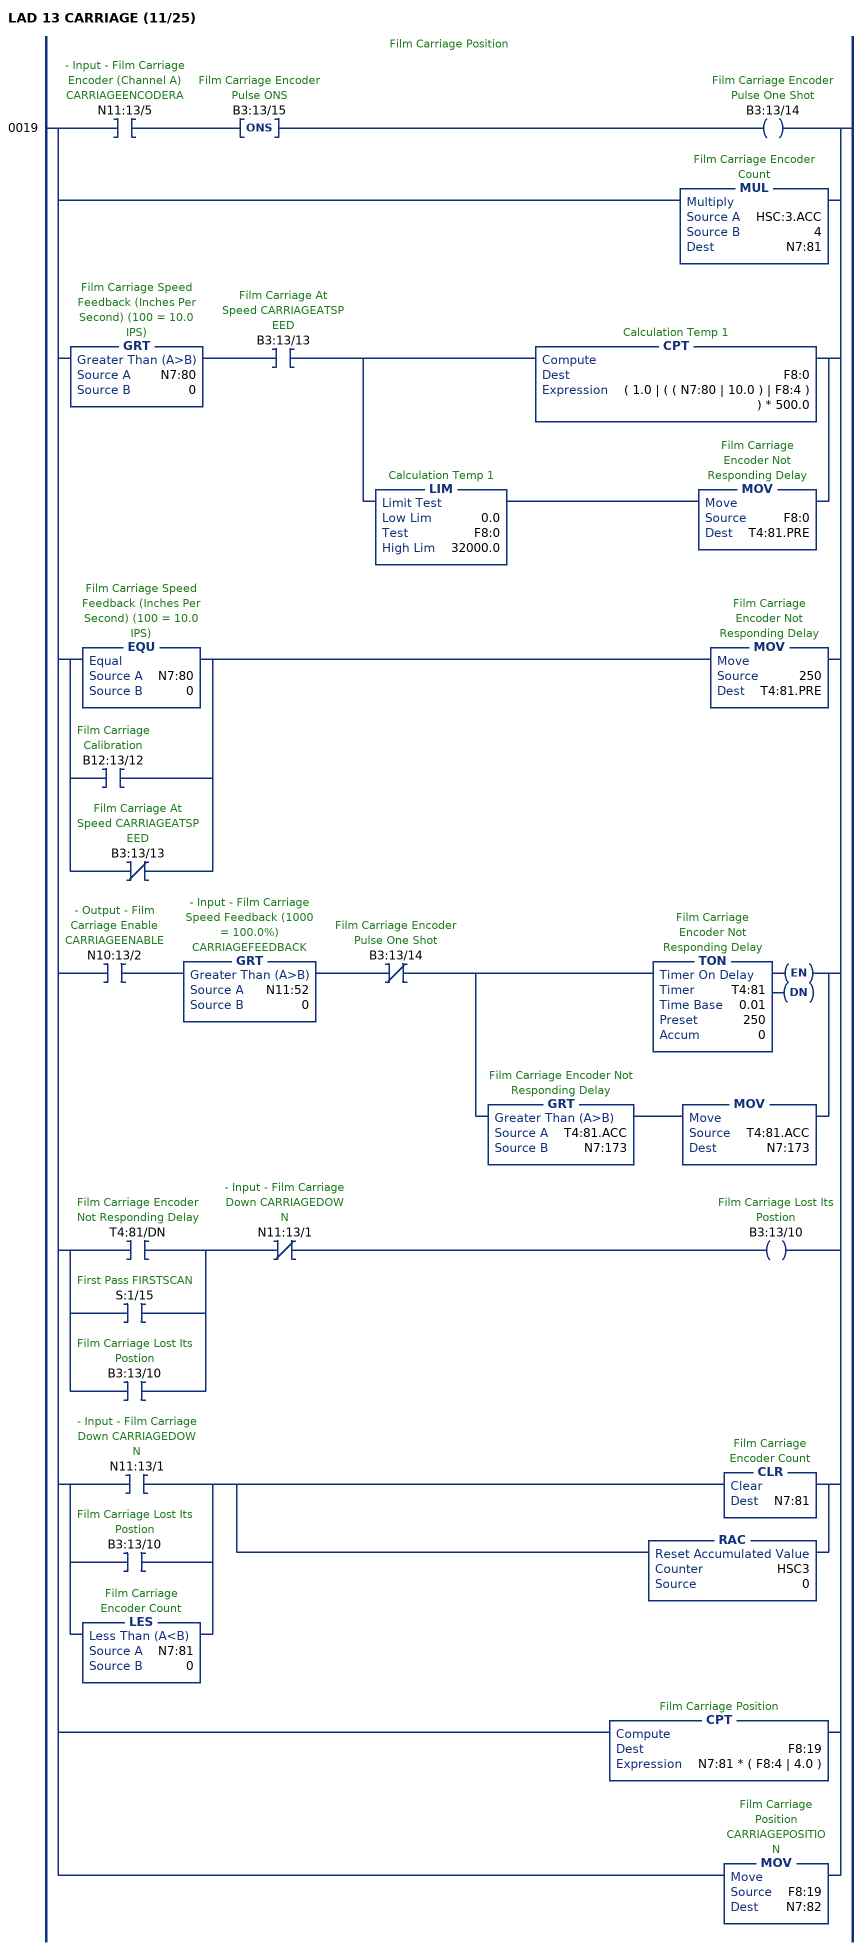
% Rung: 19 %
% Film Carriage Position %
SOR BST XIC N11:13/5 ONS B3:13/15 OTE B3:13/14 NXB MUL HSC:3.ACC 4 N7:81 NXB BST GRT N7:80 0 XIC B3:13/13 BST CPT F8:0 " ( 1.0 | ( ( N7:80 | 10.0 ) | F8:4 ) ) * 500.0 " NXB LIM 0.0 F8:0 32000.0 MOV F8:0 T4:81.PRE BND NXB BST EQU N7:80 0 NXB XIC B12:13/12 NXB XIO B3:13/13 BND MOV 250 T4:81.PRE BND NXB XIC N10:13/2 GRT N11:52 0 XIO B3:13/14 BST TON T4:81 0.01 250 0 NXB GRT T4:81.ACC N7:173 MOV T4:81.ACC N7:173 BND NXB BST XIC T4:81/DN NXB XIC S:1/15 NXB XIC B3:13/10 BND XIO N11:13/1 OTE B3:13/10 NXB BST XIC N11:13/1 NXB XIC B3:13/10 NXB LES N7:81 0 BND BST CLR N7:81 NXB RAC HSC3 0 BND NXB CPT F8:19 " N7:81 * ( F8:4 | 4.0 ) " NXB MOV F8:19 N7:82 BND EOR
%   N11:13/5  CARRIAGEENCODERA  "- Input - Film Carriage Encoder (Channel A)" %
%   B3:13/15  "Film Carriage Encoder Pulse ONS" %
%   B3:13/14  "Film Carriage Encoder Pulse One Shot" %
%   N7:81  "Film Carriage Encoder Count" %
%   N7:80  "Film Carriage Speed Feedback (Inches Per Second) (100 = 10.0 IPS)" %
%   B3:13/13  CARRIAGEATSPEED  "Film Carriage At Speed" %
%   F8:0  "Calculation Temp 1" %
%   F8:4  CARRIAGEENCODERRES  "Film Carriage Encoder Resolution (Inches Per Pulse)" %
%   T4:81  "Film Carriage Encoder Not Responding Delay" %
%   B12:13/12  "Film Carriage Calibration" %
%   N10:13/2  CARRIAGEENABLE  "- Output - Film Carriage Enable" %
%   N11:52  CARRIAGEFEEDBACK  "- Input - Film Carriage Speed Feedback (1000 = 100.0%)" %
%   S:1/15  FIRSTSCAN  "First Pass" %
%   B3:13/10  "Film Carriage Lost Its Postion" %
%   N11:13/1  CARRIAGEDOWN  "- Input - Film Carriage Down" %
%   F8:19  "Film Carriage Position" %
%   N7:82  CARRIAGEPOSITION  "Film Carriage Position" %

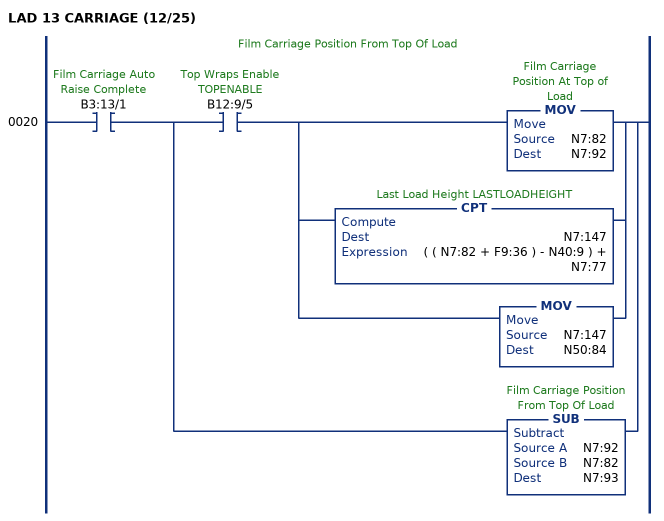
% Rung: 20 %
% Film Carriage Position From Top Of Load %
SOR XIC B3:13/1 BST XIC B12:9/5 BST MOV N7:82 N7:92 NXB CPT N7:147 " ( ( N7:82 + F9:36 ) - N40:9 ) + N7:77 " NXB MOV N7:147 N50:84 BND NXB SUB N7:92 N7:82 N7:93 BND EOR
%   B3:13/1  "Film Carriage Auto Raise Complete" %
%   B12:9/5  TOPENABLE  "Top Wraps Enable" %
%   N7:82  CARRIAGEPOSITION  "Film Carriage Position" %
%   N7:92  "Film Carriage Position At Top of Load" %
%   N7:147  LASTLOADHEIGHT  "Last Load Height" %
%   F9:36  FILMWIDTHATLOAD  "Film Width At Load" %
%   N40:9  "Current Profile Top Overwrap (Inches)" %
%   N7:77  "Carriage Pallet Grip Drive Down" %
%   N7:93  "Film Carriage Position From Top Of Load" %

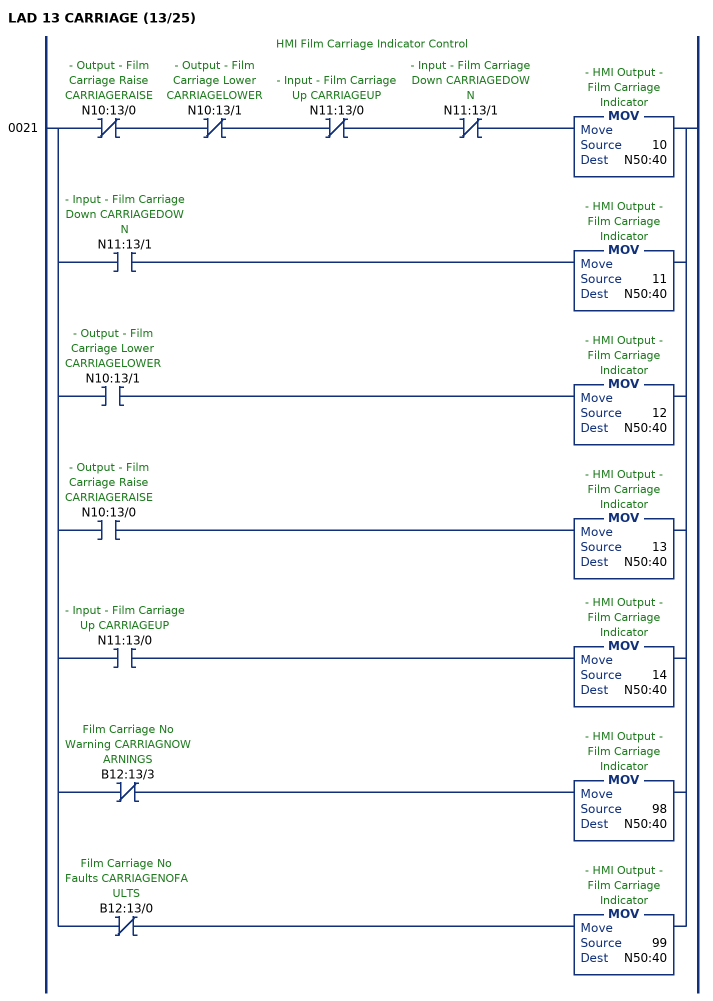
% Rung: 21 %
% HMI Film Carriage Indicator Control %
SOR BST XIO N10:13/0 XIO N10:13/1 XIO N11:13/0 XIO N11:13/1 MOV 10 N50:40 NXB XIC N11:13/1 MOV 11 N50:40 NXB XIC N10:13/1 MOV 12 N50:40 NXB XIC N10:13/0 MOV 13 N50:40 NXB XIC N11:13/0 MOV 14 N50:40 NXB XIO B12:13/3 MOV 98 N50:40 NXB XIO B12:13/0 MOV 99 N50:40 BND EOR
%   N10:13/0  CARRIAGERAISE  "- Output - Film Carriage Raise" %
%   N10:13/1  CARRIAGELOWER  "- Output - Film Carriage Lower" %
%   N11:13/0  CARRIAGEUP  "- Input - Film Carriage Up" %
%   N11:13/1  CARRIAGEDOWN  "- Input - Film Carriage Down" %
%   N50:40  "- HMI Output - Film Carriage Indicator" %
%   B12:13/3  CARRIAGNOWARNINGS  "Film Carriage No Warning" %
%   B12:13/0  CARRIAGENOFAULTS  "Film Carriage No Faults" %

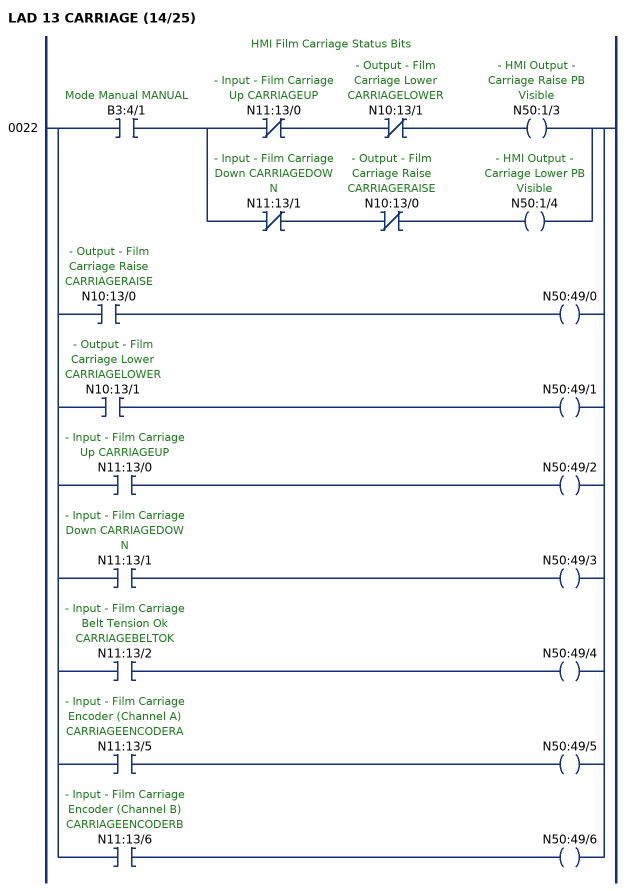
% Rung: 22 %
% HMI Film Carriage Status Bits %
SOR BST XIC B3:4/1 BST XIO N11:13/0 XIO N10:13/1 OTE N50:1/3 NXB XIO N11:13/1 XIO N10:13/0 OTE N50:1/4 BND NXB XIC N10:13/0 OTE N50:49/0 NXB XIC N10:13/1 OTE N50:49/1 NXB XIC N11:13/0 OTE N50:49/2 NXB XIC N11:13/1 OTE N50:49/3 NXB XIC N11:13/2 OTE N50:49/4 NXB XIC N11:13/5 OTE N50:49/5 NXB XIC N11:13/6 OTE N50:49/6 BND EOR
%   B3:4/1  MANUAL  "Mode Manual" %
%   N11:13/0  CARRIAGEUP  "- Input - Film Carriage Up" %
%   N10:13/1  CARRIAGELOWER  "- Output - Film Carriage Lower" %
%   N50:1/3  "- HMI Output - Carriage Raise PB Visible" %
%   N11:13/1  CARRIAGEDOWN  "- Input - Film Carriage Down" %
%   N10:13/0  CARRIAGERAISE  "- Output - Film Carriage Raise" %
%   N50:1/4  "- HMI Output - Carriage Lower PB Visible" %
%   N11:13/2  CARRIAGEBELTOK  "- Input - Film Carriage Belt Tension Ok" %
%   N11:13/5  CARRIAGEENCODERA  "- Input - Film Carriage Encoder (Channel A)" %
%   N11:13/6  CARRIAGEENCODERB  "- Input - Film Carriage Encoder (Channel B)" %

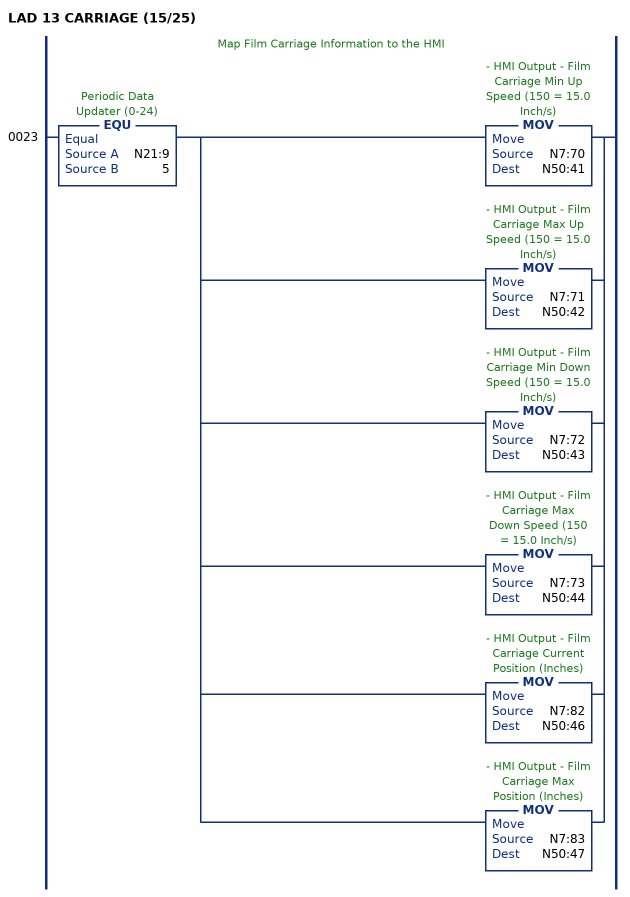
% Rung: 23 %
% Map Film Carriage Information to the HMI %
SOR EQU N21:9 5 BST MOV N7:70 N50:41 NXB MOV N7:71 N50:42 NXB MOV N7:72 N50:43 NXB MOV N7:73 N50:44 NXB MOV N7:82 N50:46 NXB MOV N7:83 N50:47 BND EOR
%   N21:9  "Periodic Data Updater (0-24)" %
%   N7:70  "Film Carriage Up Min Speed (Inches Per Second) (100 = 10.0 IPS)" %
%   N50:41  "- HMI Output - Film Carriage Min Up Speed (150 = 15.0 Inch/s)" %
%   N7:71  "Film Carriage Up Max Speed (Inches Per Second) (100 = 10.0 IPS)" %
%   N50:42  "- HMI Output - Film Carriage Max Up Speed (150 = 15.0 Inch/s)" %
%   N7:72  "Film Carriage Down Min Speed (Inches Per Second) (100 = 10.0 IPS)" %
%   N50:43  "- HMI Output - Film Carriage Min Down Speed (150 = 15.0 Inch/s)" %
%   N7:73  "Film Carriage Down Max Speed (Inches Per Second) (100 = 10.0 IPS)" %
%   N50:44  "- HMI Output - Film Carriage Max Down Speed (150 = 15.0 Inch/s)" %
%   N7:82  CARRIAGEPOSITION  "Film Carriage Position" %
%   N50:46  "- HMI Output - Film Carriage Current Position (Inches)" %
%   N7:83  CARRIAGEMAXPOSITION  "Film Carriage Max Position" %
%   N50:47  "- HMI Output - Film Carriage Max Position (Inches)" %

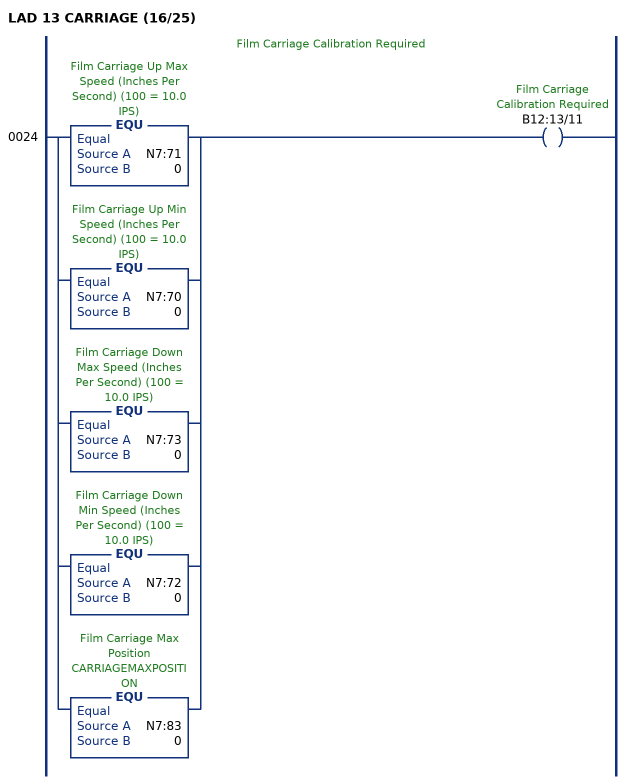
% Rung: 24 %
% Film Carriage Calibration Required %
SOR BST EQU N7:71 0 NXB EQU N7:70 0 NXB EQU N7:73 0 NXB EQU N7:72 0 NXB EQU N7:83 0 BND OTE B12:13/11 EOR
%   N7:71  "Film Carriage Up Max Speed (Inches Per Second) (100 = 10.0 IPS)" %
%   N7:70  "Film Carriage Up Min Speed (Inches Per Second) (100 = 10.0 IPS)" %
%   N7:73  "Film Carriage Down Max Speed (Inches Per Second) (100 = 10.0 IPS)" %
%   N7:72  "Film Carriage Down Min Speed (Inches Per Second) (100 = 10.0 IPS)" %
%   N7:83  CARRIAGEMAXPOSITION  "Film Carriage Max Position" %
%   B12:13/11  "Film Carriage Calibration Required" %

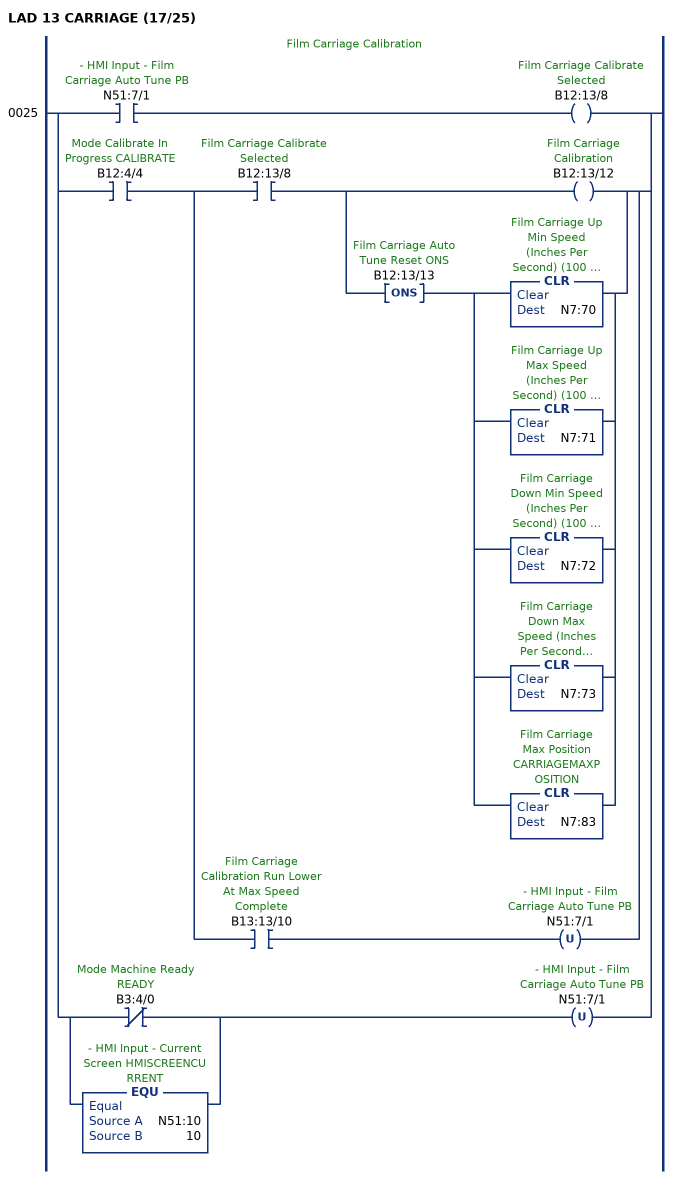
% Rung: 25 %
% Film Carriage Calibration %
SOR BST XIC N51:7/1 OTE B12:13/8 NXB XIC B12:4/4 BST XIC B12:13/8 BST OTE B12:13/12 NXB ONS B12:13/13 BST CLR N7:70 NXB CLR N7:71 NXB CLR N7:72 NXB CLR N7:73 NXB CLR N7:83 BND BND NXB XIC B13:13/10 OTU N51:7/1 BND NXB BST XIO B3:4/0 NXB EQU N51:10 10 BND OTU N51:7/1 BND EOR
%   N51:7/1  "- HMI Input - Film Carriage Auto Tune PB" %
%   B12:13/8  "Film Carriage Calibrate Selected" %
%   B12:4/4  CALIBRATE  "Mode Calibrate In Progress" %
%   B12:13/12  "Film Carriage Calibration" %
%   B12:13/13  "Film Carriage Auto Tune Reset ONS" %
%   N7:70  "Film Carriage Up Min Speed (Inches Per Second) (100 = 10.0 IPS)" %
%   N7:71  "Film Carriage Up Max Speed (Inches Per Second) (100 = 10.0 IPS)" %
%   N7:72  "Film Carriage Down Min Speed (Inches Per Second) (100 = 10.0 IPS)" %
%   N7:73  "Film Carriage Down Max Speed (Inches Per Second) (100 = 10.0 IPS)" %
%   N7:83  CARRIAGEMAXPOSITION  "Film Carriage Max Position" %
%   B13:13/10  "Film Carriage Calibration Run Lower At Max Speed Complete" %
%   B3:4/0  READY  "Mode Machine Ready" %
%   N51:10  HMISCREENCURRENT  "- HMI Input - Current Screen" %

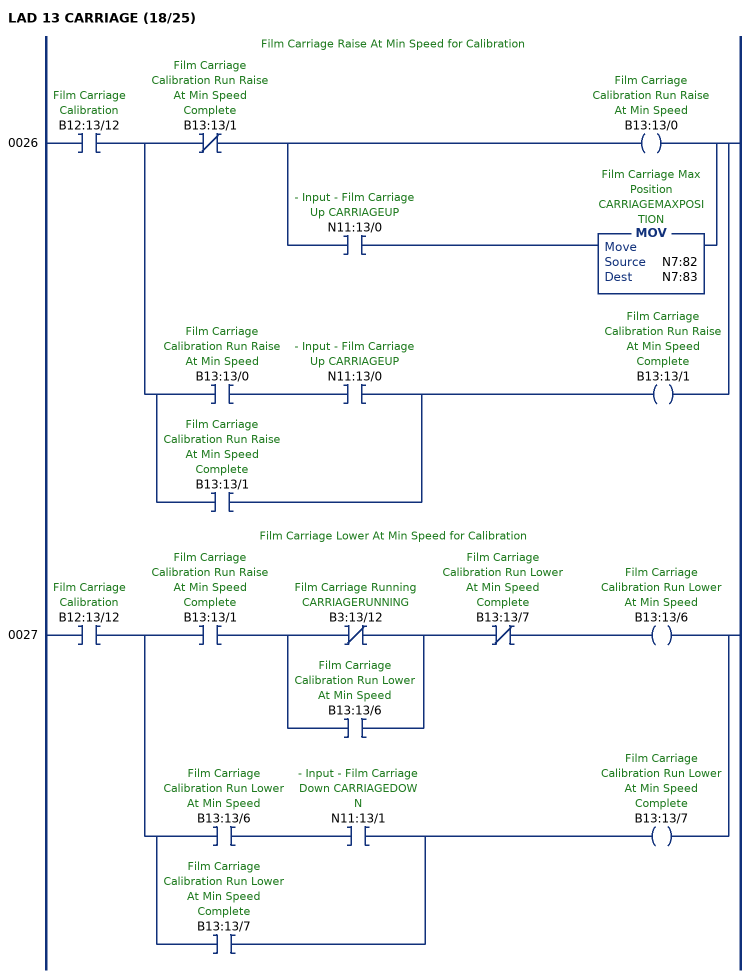
% Rung: 26 %
% Film Carriage Raise At Min Speed for Calibration %
SOR XIC B12:13/12 BST XIO B13:13/1 BST OTE B13:13/0 NXB XIC N11:13/0 MOV N7:82 N7:83 BND NXB BST XIC B13:13/0 XIC N11:13/0 NXB XIC B13:13/1 BND OTE B13:13/1 BND EOR
%   B12:13/12  "Film Carriage Calibration" %
%   B13:13/1  "Film Carriage Calibration Run Raise At Min Speed Complete" %
%   B13:13/0  "Film Carriage Calibration Run Raise At Min Speed" %
%   N11:13/0  CARRIAGEUP  "- Input - Film Carriage Up" %
%   N7:82  CARRIAGEPOSITION  "Film Carriage Position" %
%   N7:83  CARRIAGEMAXPOSITION  "Film Carriage Max Position" %
% Rung: 27 %
% Film Carriage Lower At Min Speed for Calibration %
SOR XIC B12:13/12 BST XIC B13:13/1 BST XIO B3:13/12 NXB XIC B13:13/6 BND XIO B13:13/7 OTE B13:13/6 NXB BST XIC B13:13/6 XIC N11:13/1 NXB XIC B13:13/7 BND OTE B13:13/7 BND EOR
%   B12:13/12  "Film Carriage Calibration" %
%   B13:13/1  "Film Carriage Calibration Run Raise At Min Speed Complete" %
%   B3:13/12  CARRIAGERUNNING  "Film Carriage Running" %
%   B13:13/6  "Film Carriage Calibration Run Lower At Min Speed" %
%   B13:13/7  "Film Carriage Calibration Run Lower At Min Speed Complete" %
%   N11:13/1  CARRIAGEDOWN  "- Input - Film Carriage Down" %

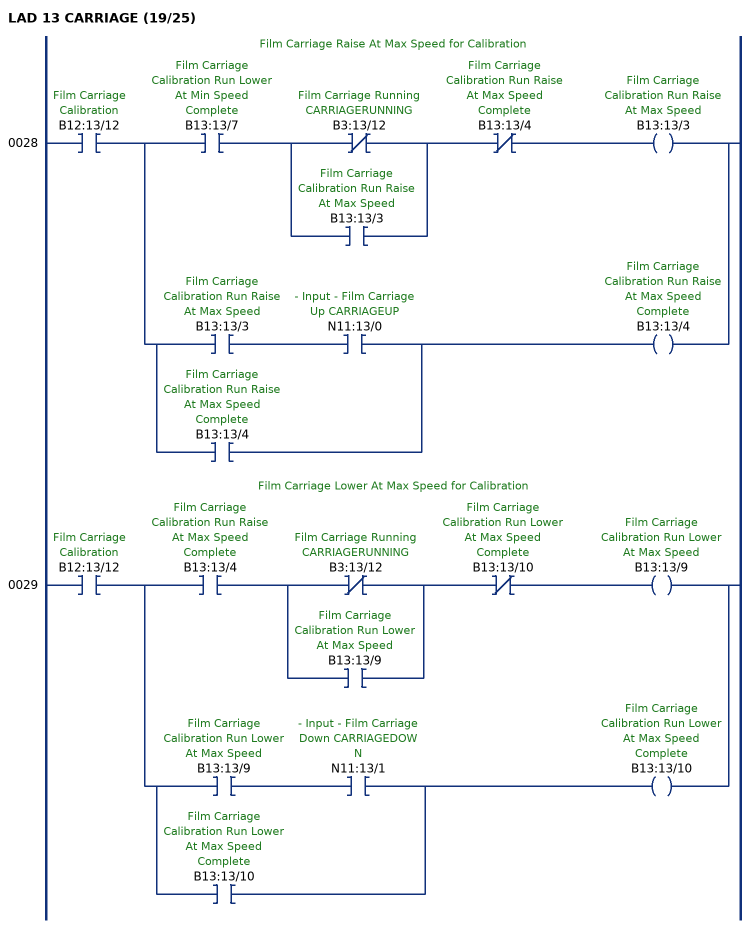
% Rung: 28 %
% Film Carriage Raise At Max Speed for Calibration %
SOR XIC B12:13/12 BST XIC B13:13/7 BST XIO B3:13/12 NXB XIC B13:13/3 BND XIO B13:13/4 OTE B13:13/3 NXB BST XIC B13:13/3 XIC N11:13/0 NXB XIC B13:13/4 BND OTE B13:13/4 BND EOR
%   B12:13/12  "Film Carriage Calibration" %
%   B13:13/7  "Film Carriage Calibration Run Lower At Min Speed Complete" %
%   B3:13/12  CARRIAGERUNNING  "Film Carriage Running" %
%   B13:13/3  "Film Carriage Calibration Run Raise At Max Speed" %
%   B13:13/4  "Film Carriage Calibration Run Raise At Max Speed Complete" %
%   N11:13/0  CARRIAGEUP  "- Input - Film Carriage Up" %
% Rung: 29 %
% Film Carriage Lower At Max Speed for Calibration %
SOR XIC B12:13/12 BST XIC B13:13/4 BST XIO B3:13/12 NXB XIC B13:13/9 BND XIO B13:13/10 OTE B13:13/9 NXB BST XIC B13:13/9 XIC N11:13/1 NXB XIC B13:13/10 BND OTE B13:13/10 BND EOR
%   B12:13/12  "Film Carriage Calibration" %
%   B13:13/4  "Film Carriage Calibration Run Raise At Max Speed Complete" %
%   B3:13/12  CARRIAGERUNNING  "Film Carriage Running" %
%   B13:13/9  "Film Carriage Calibration Run Lower At Max Speed" %
%   B13:13/10  "Film Carriage Calibration Run Lower At Max Speed Complete" %
%   N11:13/1  CARRIAGEDOWN  "- Input - Film Carriage Down" %

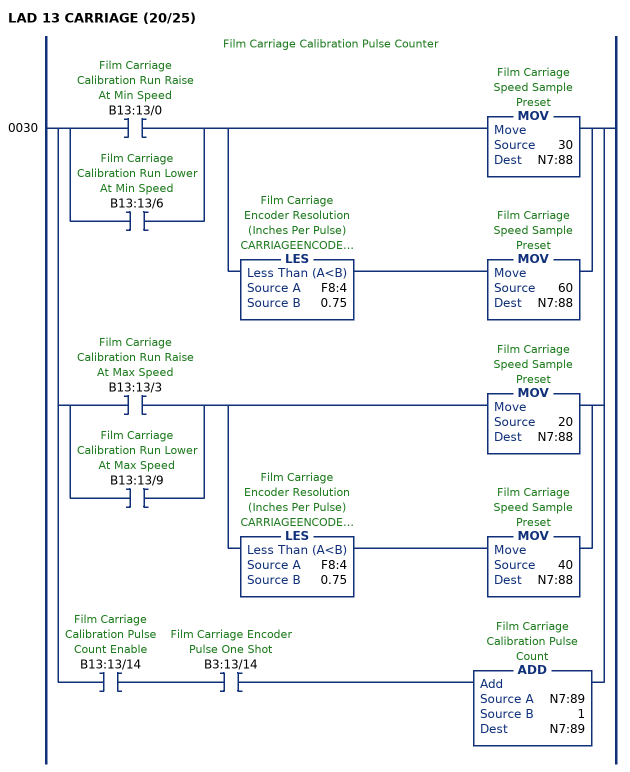
% Rung: 30 %
% Film Carriage Calibration Pulse Counter %
SOR BST BST XIC B13:13/0 NXB XIC B13:13/6 BND BST MOV 30 N7:88 NXB LES F8:4 0.75 MOV 60 N7:88 BND NXB BST XIC B13:13/3 NXB XIC B13:13/9 BND BST MOV 20 N7:88 NXB LES F8:4 0.75 MOV 40 N7:88 BND NXB XIC B13:13/14 XIC B3:13/14 ADD N7:89 1 N7:89 BND EOR
%   B13:13/0  "Film Carriage Calibration Run Raise At Min Speed" %
%   B13:13/6  "Film Carriage Calibration Run Lower At Min Speed" %
%   N7:88  "Film Carriage Speed Sample Preset" %
%   F8:4  CARRIAGEENCODERRES  "Film Carriage Encoder Resolution (Inches Per Pulse)" %
%   B13:13/3  "Film Carriage Calibration Run Raise At Max Speed" %
%   B13:13/9  "Film Carriage Calibration Run Lower At Max Speed" %
%   B13:13/14  "Film Carriage Calibration Pulse Count Enable" %
%   B3:13/14  "Film Carriage Encoder Pulse One Shot" %
%   N7:89  "Film Carriage Calibration Pulse Count" %

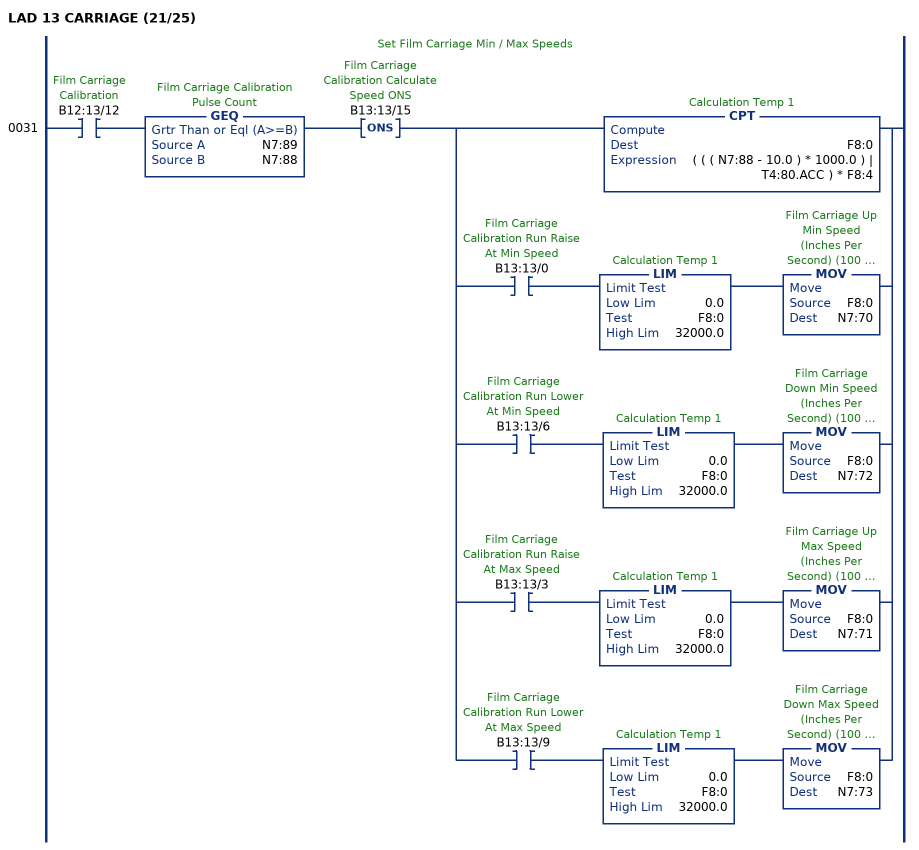
% Rung: 31 %
% Set Film Carriage Min / Max Speeds %
SOR XIC B12:13/12 GEQ N7:89 N7:88 ONS B13:13/15 BST CPT F8:0 " ( ( ( N7:88 - 10.0 ) * 1000.0 ) | T4:80.ACC ) * F8:4 " NXB XIC B13:13/0 LIM 0.0 F8:0 32000.0 MOV F8:0 N7:70 NXB XIC B13:13/6 LIM 0.0 F8:0 32000.0 MOV F8:0 N7:72 NXB XIC B13:13/3 LIM 0.0 F8:0 32000.0 MOV F8:0 N7:71 NXB XIC B13:13/9 LIM 0.0 F8:0 32000.0 MOV F8:0 N7:73 BND EOR
%   B12:13/12  "Film Carriage Calibration" %
%   N7:89  "Film Carriage Calibration Pulse Count" %
%   N7:88  "Film Carriage Speed Sample Preset" %
%   B13:13/15  "Film Carriage Calibration Calculate Speed ONS" %
%   F8:0  "Calculation Temp 1" %
%   T4:80  "Film Carriage Calibration Time" %
%   F8:4  CARRIAGEENCODERRES  "Film Carriage Encoder Resolution (Inches Per Pulse)" %
%   B13:13/0  "Film Carriage Calibration Run Raise At Min Speed" %
%   N7:70  "Film Carriage Up Min Speed (Inches Per Second) (100 = 10.0 IPS)" %
%   B13:13/6  "Film Carriage Calibration Run Lower At Min Speed" %
%   N7:72  "Film Carriage Down Min Speed (Inches Per Second) (100 = 10.0 IPS)" %
%   B13:13/3  "Film Carriage Calibration Run Raise At Max Speed" %
%   N7:71  "Film Carriage Up Max Speed (Inches Per Second) (100 = 10.0 IPS)" %
%   B13:13/9  "Film Carriage Calibration Run Lower At Max Speed" %
%   N7:73  "Film Carriage Down Max Speed (Inches Per Second) (100 = 10.0 IPS)" %

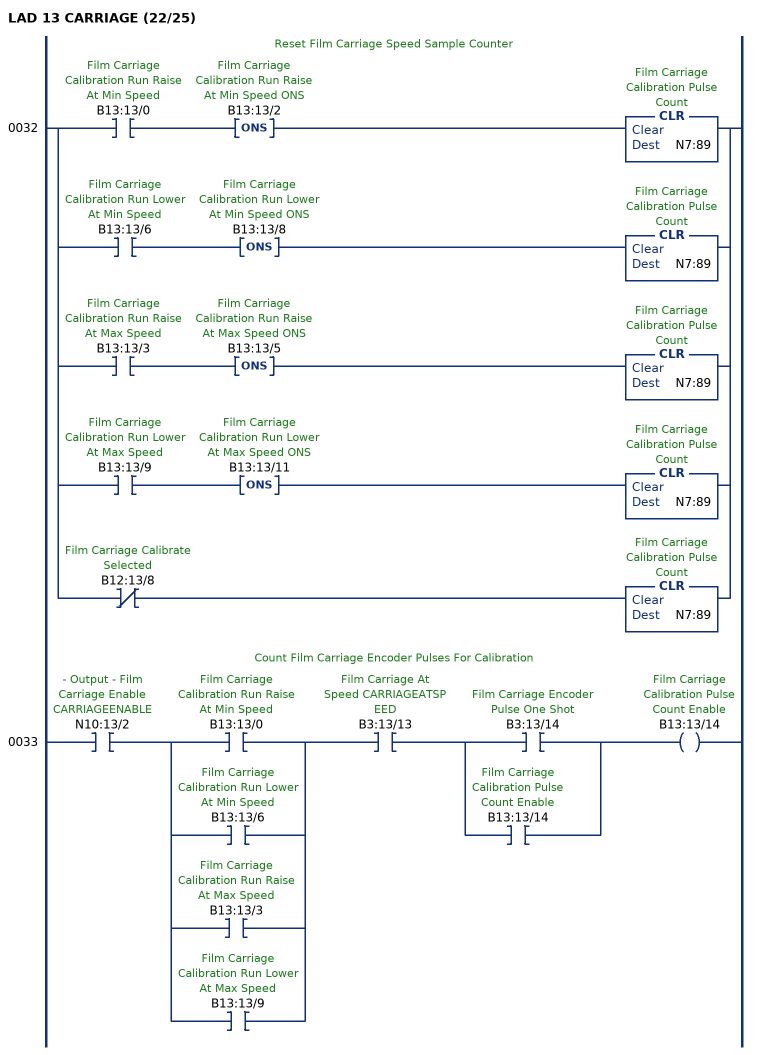
% Rung: 32 %
% Reset Film Carriage Speed Sample Counter %
SOR BST XIC B13:13/0 ONS B13:13/2 CLR N7:89 NXB XIC B13:13/6 ONS B13:13/8 CLR N7:89 NXB XIC B13:13/3 ONS B13:13/5 CLR N7:89 NXB XIC B13:13/9 ONS B13:13/11 CLR N7:89 NXB XIO B12:13/8 CLR N7:89 BND EOR
%   B13:13/0  "Film Carriage Calibration Run Raise At Min Speed" %
%   B13:13/2  "Film Carriage Calibration Run Raise At Min Speed ONS" %
%   N7:89  "Film Carriage Calibration Pulse Count" %
%   B13:13/6  "Film Carriage Calibration Run Lower At Min Speed" %
%   B13:13/8  "Film Carriage Calibration Run Lower At Min Speed ONS" %
%   B13:13/3  "Film Carriage Calibration Run Raise At Max Speed" %
%   B13:13/5  "Film Carriage Calibration Run Raise At Max Speed ONS" %
%   B13:13/9  "Film Carriage Calibration Run Lower At Max Speed" %
%   B13:13/11  "Film Carriage Calibration Run Lower At Max Speed ONS" %
%   B12:13/8  "Film Carriage Calibrate Selected" %
% Rung: 33 %
% Count Film Carriage Encoder Pulses For Calibration %
SOR XIC N10:13/2 BST XIC B13:13/0 NXB XIC B13:13/6 NXB XIC B13:13/3 NXB XIC B13:13/9 BND XIC B3:13/13 BST XIC B3:13/14 NXB XIC B13:13/14 BND OTE B13:13/14 EOR
%   N10:13/2  CARRIAGEENABLE  "- Output - Film Carriage Enable" %
%   B13:13/0  "Film Carriage Calibration Run Raise At Min Speed" %
%   B13:13/6  "Film Carriage Calibration Run Lower At Min Speed" %
%   B13:13/3  "Film Carriage Calibration Run Raise At Max Speed" %
%   B13:13/9  "Film Carriage Calibration Run Lower At Max Speed" %
%   B3:13/13  CARRIAGEATSPEED  "Film Carriage At Speed" %
%   B3:13/14  "Film Carriage Encoder Pulse One Shot" %
%   B13:13/14  "Film Carriage Calibration Pulse Count Enable" %

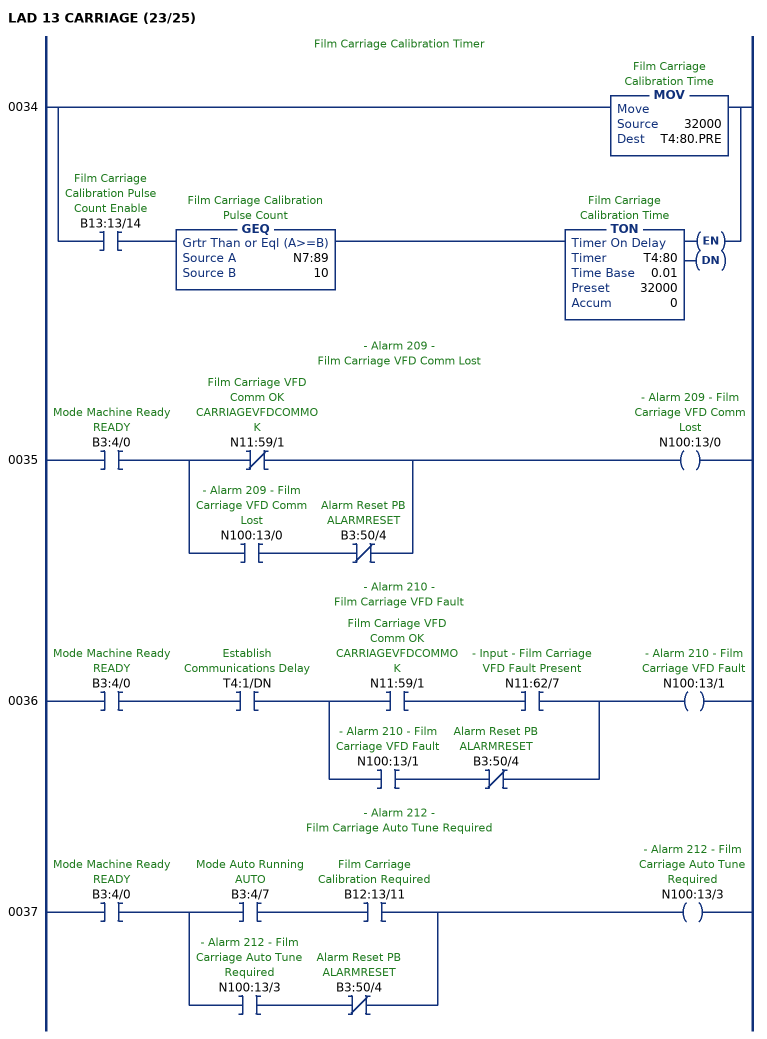
% Rung: 34 %
% Film Carriage Calibration Timer %
SOR BST MOV 32000 T4:80.PRE NXB XIC B13:13/14 GEQ N7:89 10 TON T4:80 0.01 32000 0 BND EOR
%   T4:80  "Film Carriage Calibration Time" %
%   B13:13/14  "Film Carriage Calibration Pulse Count Enable" %
%   N7:89  "Film Carriage Calibration Pulse Count" %
% Rung: 35 %
% - Alarm 209 -
% 
% Film Carriage VFD Comm Lost %
SOR XIC B3:4/0 BST XIO N11:59/1 NXB XIC N100:13/0 XIO B3:50/4 BND OTE N100:13/0 EOR
%   B3:4/0  READY  "Mode Machine Ready" %
%   N11:59/1  CARRIAGEVFDCOMMOK  "Film Carriage VFD Comm OK" %
%   N100:13/0  "- Alarm 209 - Film Carriage VFD Comm Lost" %
%   B3:50/4  ALARMRESET  "Alarm Reset PB" %
% Rung: 36 %
% - Alarm 210 -
% 
% Film Carriage VFD Fault %
SOR XIC B3:4/0 XIC T4:1/DN BST XIC N11:59/1 XIC N11:62/7 NXB XIC N100:13/1 XIO B3:50/4 BND OTE N100:13/1 EOR
%   B3:4/0  READY  "Mode Machine Ready" %
%   T4:1  "Establish Communications Delay" %
%   N11:59/1  CARRIAGEVFDCOMMOK  "Film Carriage VFD Comm OK" %
%   N11:62/7  "- Input - Film Carriage VFD Fault Present" %
%   N100:13/1  "- Alarm 210 - Film Carriage VFD Fault" %
%   B3:50/4  ALARMRESET  "Alarm Reset PB" %
% Rung: 37 %
% - Alarm 212 -
% 
% Film Carriage Auto Tune Required %
SOR XIC B3:4/0 BST XIC B3:4/7 XIC B12:13/11 NXB XIC N100:13/3 XIO B3:50/4 BND OTE N100:13/3 EOR
%   B3:4/0  READY  "Mode Machine Ready" %
%   B3:4/7  AUTO  "Mode Auto Running" %
%   B12:13/11  "Film Carriage Calibration Required" %
%   N100:13/3  "- Alarm 212 - Film Carriage Auto Tune Required" %
%   B3:50/4  ALARMRESET  "Alarm Reset PB" %

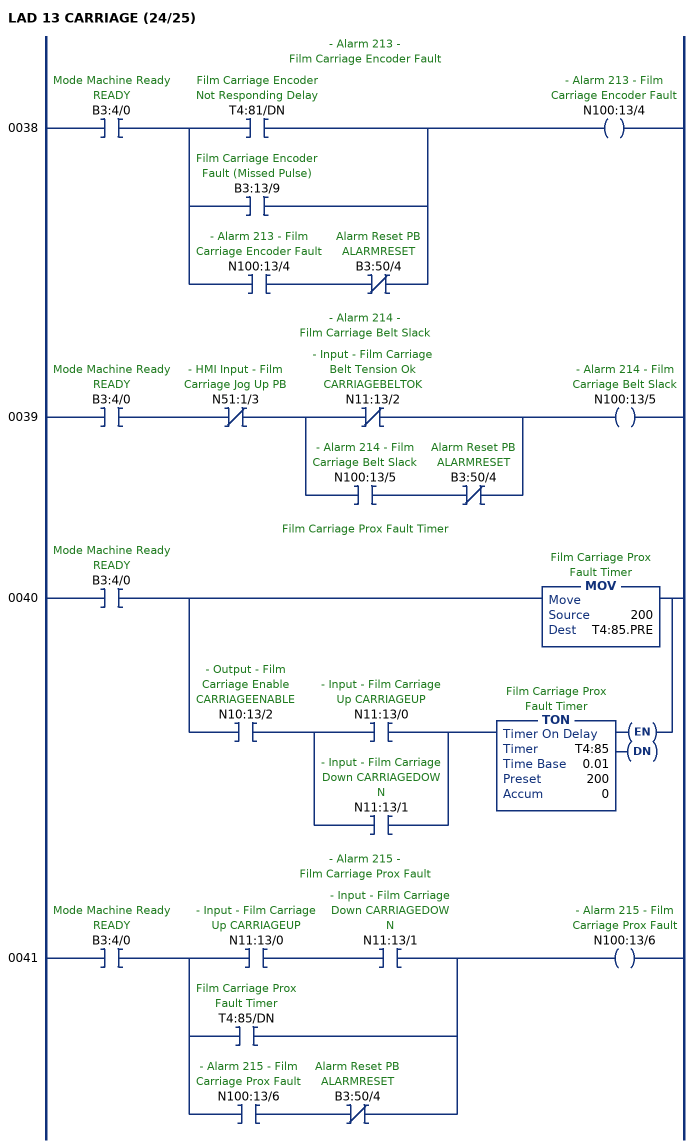
% Rung: 38 %
% - Alarm 213 -
% 
% Film Carriage Encoder Fault %
SOR XIC B3:4/0 BST XIC T4:81/DN NXB XIC B3:13/9 NXB XIC N100:13/4 XIO B3:50/4 BND OTE N100:13/4 EOR
%   B3:4/0  READY  "Mode Machine Ready" %
%   T4:81  "Film Carriage Encoder Not Responding Delay" %
%   B3:13/9  "Film Carriage Encoder Fault (Missed Pulse)" %
%   N100:13/4  "- Alarm 213 - Film Carriage Encoder Fault" %
%   B3:50/4  ALARMRESET  "Alarm Reset PB" %
% Rung: 39 %
% - Alarm 214 -
% 
% Film Carriage Belt Slack %
SOR XIC B3:4/0 XIO N51:1/3 BST XIO N11:13/2 NXB XIC N100:13/5 XIO B3:50/4 BND OTE N100:13/5 EOR
%   B3:4/0  READY  "Mode Machine Ready" %
%   N51:1/3  "- HMI Input - Film Carriage Jog Up PB" %
%   N11:13/2  CARRIAGEBELTOK  "- Input - Film Carriage Belt Tension Ok" %
%   N100:13/5  "- Alarm 214 - Film Carriage Belt Slack" %
%   B3:50/4  ALARMRESET  "Alarm Reset PB" %
% Rung: 40 %
% Film Carriage Prox Fault Timer %
SOR XIC B3:4/0 BST MOV 200 T4:85.PRE NXB XIC N10:13/2 BST XIC N11:13/0 NXB XIC N11:13/1 BND TON T4:85 0.01 200 0 BND EOR
%   B3:4/0  READY  "Mode Machine Ready" %
%   T4:85  "Film Carriage Prox Fault Timer" %
%   N10:13/2  CARRIAGEENABLE  "- Output - Film Carriage Enable" %
%   N11:13/0  CARRIAGEUP  "- Input - Film Carriage Up" %
%   N11:13/1  CARRIAGEDOWN  "- Input - Film Carriage Down" %
% Rung: 41 %
% - Alarm 215 -
% 
% Film Carriage Prox Fault %
SOR XIC B3:4/0 BST XIC N11:13/0 XIC N11:13/1 NXB XIC T4:85/DN NXB XIC N100:13/6 XIO B3:50/4 BND OTE N100:13/6 EOR
%   B3:4/0  READY  "Mode Machine Ready" %
%   N11:13/0  CARRIAGEUP  "- Input - Film Carriage Up" %
%   N11:13/1  CARRIAGEDOWN  "- Input - Film Carriage Down" %
%   T4:85  "Film Carriage Prox Fault Timer" %
%   N100:13/6  "- Alarm 215 - Film Carriage Prox Fault" %
%   B3:50/4  ALARMRESET  "Alarm Reset PB" %

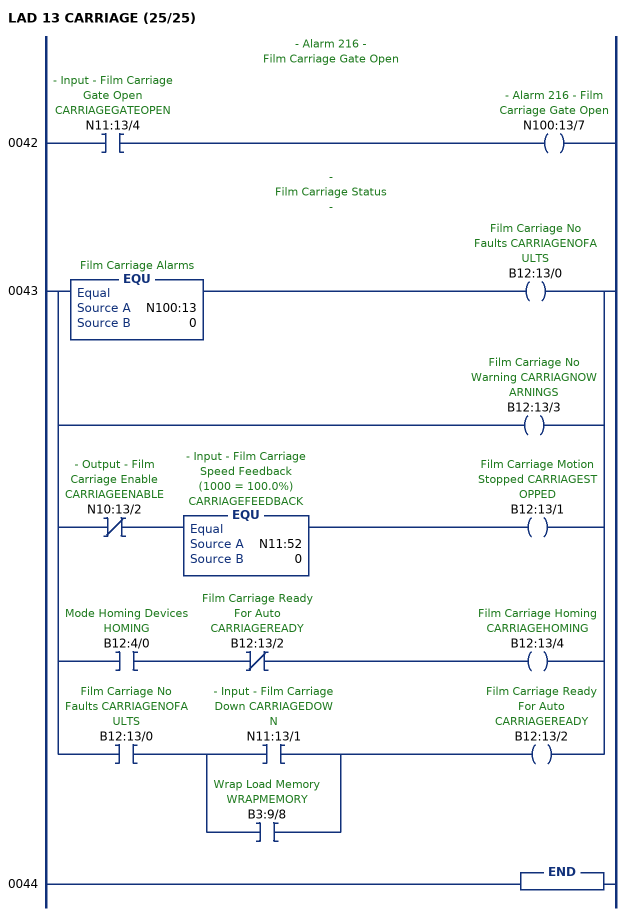
% Rung: 42 %
% - Alarm 216 -
% 
% Film Carriage Gate Open %
SOR XIC N11:13/4 OTE N100:13/7 EOR
%   N11:13/4  CARRIAGEGATEOPEN  "- Input - Film Carriage Gate Open" %
%   N100:13/7  "- Alarm 216 - Film Carriage Gate Open" %
% Rung: 43 %
% -
% 
% Film Carriage Status
% 
% - %
SOR BST EQU N100:13 0 OTE B12:13/0 NXB OTE B12:13/3 NXB XIO N10:13/2 EQU N11:52 0 OTE B12:13/1 NXB XIC B12:4/0 XIO B12:13/2 OTE B12:13/4 NXB XIC B12:13/0 BST XIC N11:13/1 NXB XIC B3:9/8 BND OTE B12:13/2 BND EOR
%   N100:13  "Film Carriage Alarms" %
%   B12:13/0  CARRIAGENOFAULTS  "Film Carriage No Faults" %
%   B12:13/3  CARRIAGNOWARNINGS  "Film Carriage No Warning" %
%   N10:13/2  CARRIAGEENABLE  "- Output - Film Carriage Enable" %
%   N11:52  CARRIAGEFEEDBACK  "- Input - Film Carriage Speed Feedback (1000 = 100.0%)" %
%   B12:13/1  CARRIAGESTOPPED  "Film Carriage Motion Stopped" %
%   B12:4/0  HOMING  "Mode Homing Devices" %
%   B12:13/2  CARRIAGEREADY  "Film Carriage Ready For Auto" %
%   B12:13/4  CARRIAGEHOMING  "Film Carriage Homing" %
%   N11:13/1  CARRIAGEDOWN  "- Input - Film Carriage Down" %
%   B3:9/8  WRAPMEMORY  "Wrap Load Memory" %
% Rung: 44 %
SOR END EOR

LADDER 14 "MPS"
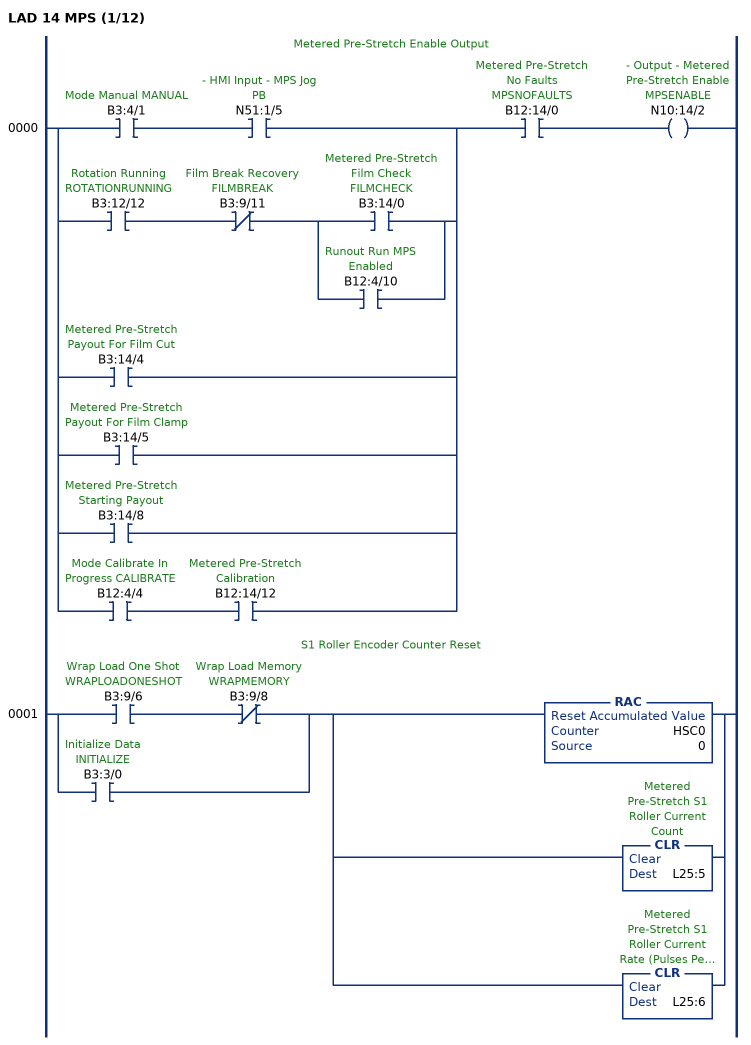
% Rung: 0 %
% Metered Pre-Stretch Enable Output %
SOR BST XIC B3:4/1 XIC N51:1/5 NXB XIC B3:12/12 XIO B3:9/11 BST XIC B3:14/0 NXB XIC B12:4/10 BND NXB XIC B3:14/4 NXB XIC B3:14/5 NXB XIC B3:14/8 NXB XIC B12:4/4 XIC B12:14/12 BND XIC B12:14/0 OTE N10:14/2 EOR
%   B3:4/1  MANUAL  "Mode Manual" %
%   N51:1/5  "- HMI Input - MPS Jog PB" %
%   B3:12/12  ROTATIONRUNNING  "Rotation Running" %
%   B3:9/11  FILMBREAK  "Film Break Recovery" %
%   B3:14/0  FILMCHECK  "Metered Pre-Stretch Film Check" %
%   B12:4/10  "Runout Run MPS Enabled" %
%   B3:14/4  "Metered Pre-Stretch Payout For Film Cut" %
%   B3:14/5  "Metered Pre-Stretch Payout For Film Clamp" %
%   B3:14/8  "Metered Pre-Stretch Starting Payout" %
%   B12:4/4  CALIBRATE  "Mode Calibrate In Progress" %
%   B12:14/12  "Metered Pre-Stretch Calibration" %
%   B12:14/0  MPSNOFAULTS  "Metered Pre-Stretch No Faults" %
%   N10:14/2  MPSENABLE  "- Output - Metered Pre-Stretch Enable" %
% Rung: 1 %
% S1 Roller Encoder Counter Reset %
SOR BST XIC B3:9/6 XIO B3:9/8 NXB XIC B3:3/0 BND BST RAC HSC0 0 NXB CLR L25:5 NXB CLR L25:6 BND EOR
%   B3:9/6  WRAPLOADONESHOT  "Wrap Load One Shot" %
%   B3:9/8  WRAPMEMORY  "Wrap Load Memory" %
%   B3:3/0  INITIALIZE  "Initialize Data" %
%   L25:5  "Metered Pre-Stretch S1 Roller Current Count" %
%   L25:6  "Metered Pre-Stretch S1 Roller Current Rate (Pulses Per Second)" %

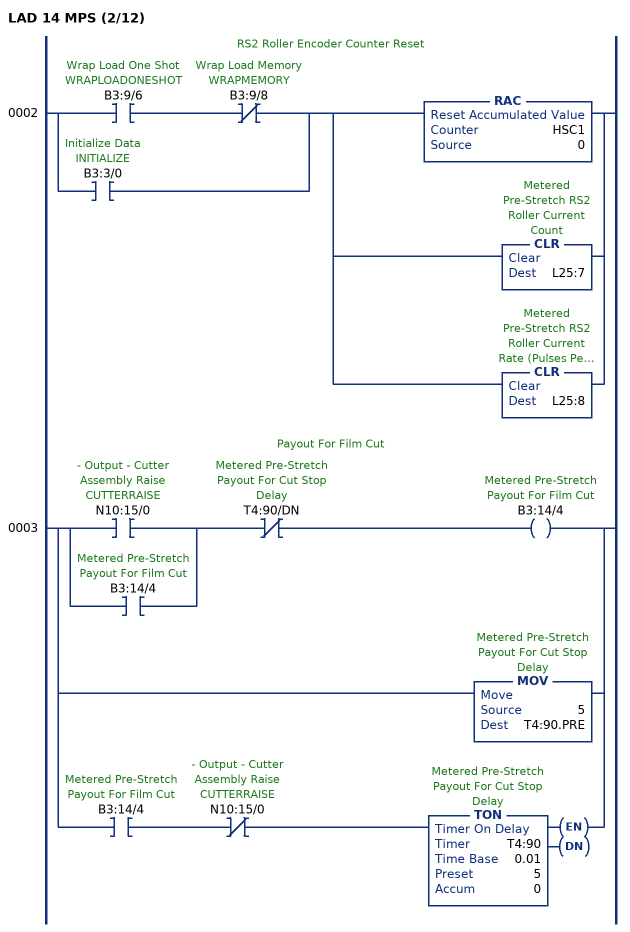
% Rung: 2 %
% RS2 Roller Encoder Counter Reset %
SOR BST XIC B3:9/6 XIO B3:9/8 NXB XIC B3:3/0 BND BST RAC HSC1 0 NXB CLR L25:7 NXB CLR L25:8 BND EOR
%   B3:9/6  WRAPLOADONESHOT  "Wrap Load One Shot" %
%   B3:9/8  WRAPMEMORY  "Wrap Load Memory" %
%   B3:3/0  INITIALIZE  "Initialize Data" %
%   L25:7  "Metered Pre-Stretch RS2 Roller Current Count" %
%   L25:8  "Metered Pre-Stretch RS2 Roller Current Rate (Pulses Per Second)" %
% Rung: 3 %
% Payout For Film Cut %
SOR BST BST XIC N10:15/0 NXB XIC B3:14/4 BND XIO T4:90/DN OTE B3:14/4 NXB MOV 5 T4:90.PRE NXB XIC B3:14/4 XIO N10:15/0 TON T4:90 0.01 5 0 BND EOR
%   N10:15/0  CUTTERRAISE  "- Output - Cutter Assembly Raise" %
%   B3:14/4  "Metered Pre-Stretch Payout For Film Cut" %
%   T4:90  "Metered Pre-Stretch Payout For Cut Stop Delay" %

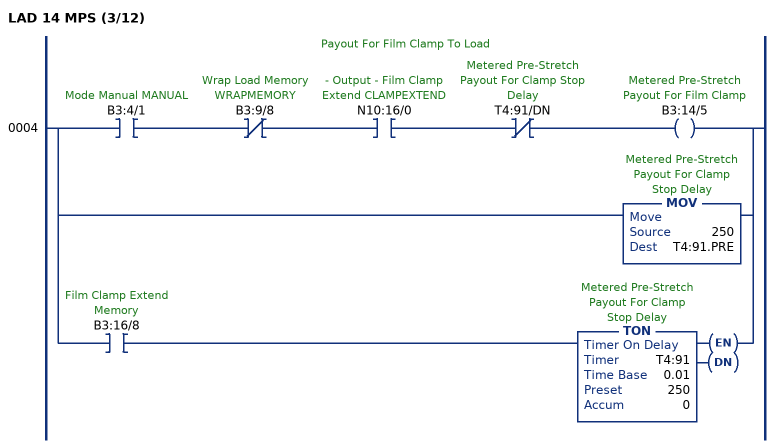
% Rung: 4 %
% Payout For Film Clamp To Load %
SOR BST XIC B3:4/1 XIO B3:9/8 XIC N10:16/0 XIO T4:91/DN OTE B3:14/5 NXB MOV 250 T4:91.PRE NXB XIC B3:16/8 TON T4:91 0.01 250 0 BND EOR
%   B3:4/1  MANUAL  "Mode Manual" %
%   B3:9/8  WRAPMEMORY  "Wrap Load Memory" %
%   N10:16/0  CLAMPEXTEND  "- Output - Film Clamp Extend" %
%   T4:91  "Metered Pre-Stretch Payout For Clamp Stop Delay" %
%   B3:14/5  "Metered Pre-Stretch Payout For Film Clamp" %
%   B3:16/8  "Film Clamp Extend Memory" %

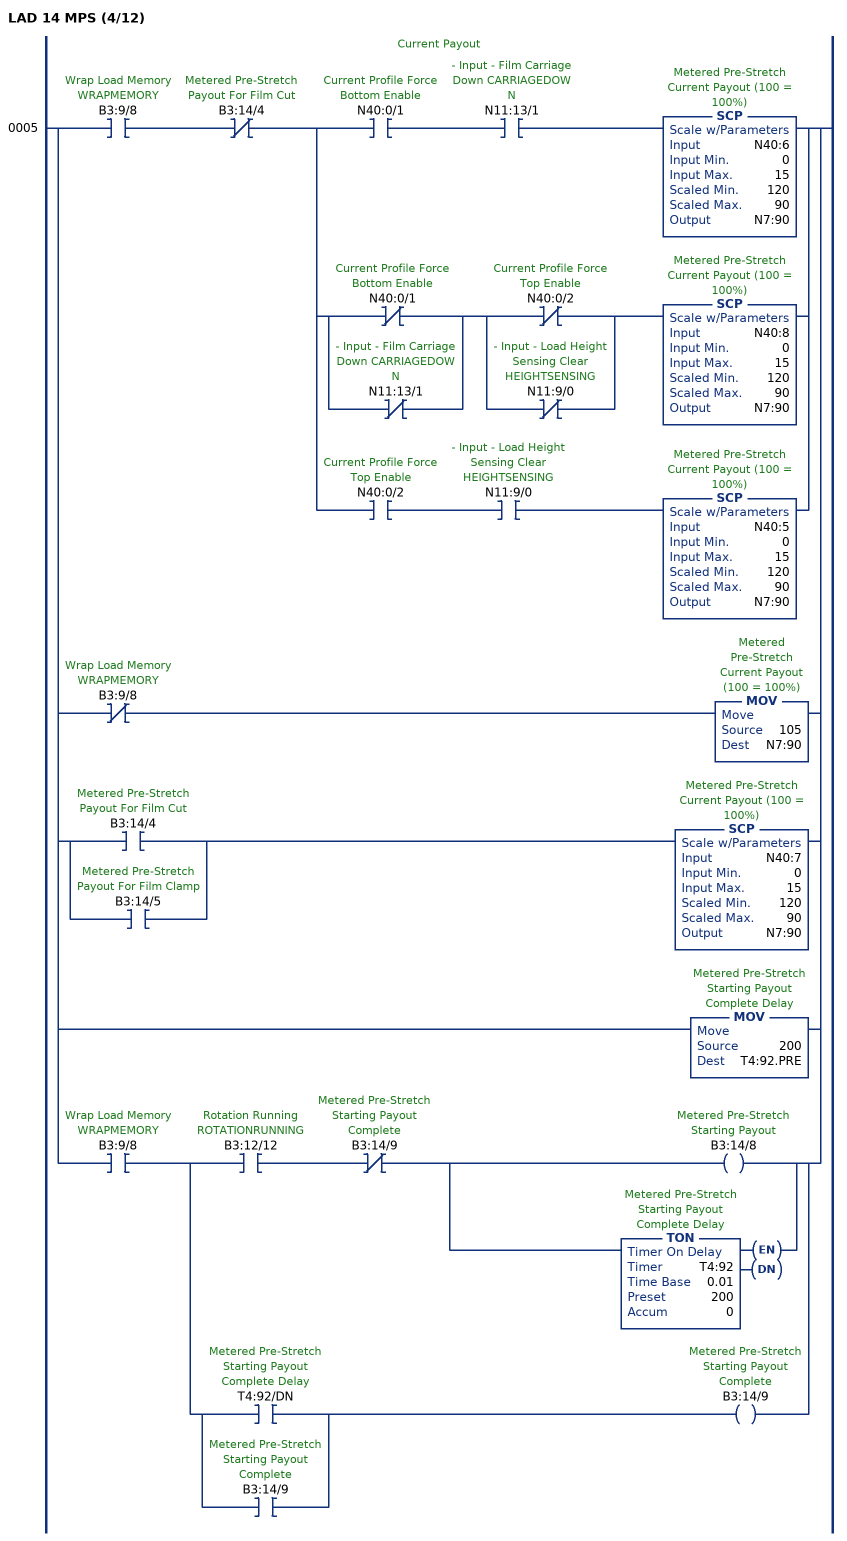
% Rung: 5 %
% Current Payout %
SOR BST XIC B3:9/8 XIO B3:14/4 BST XIC N40:0/1 XIC N11:13/1 SCP N40:6 0 15 120 90 N7:90 NXB BST XIO N40:0/1 NXB XIO N11:13/1 BND BST XIO N40:0/2 NXB XIO N11:9/0 BND SCP N40:8 0 15 120 90 N7:90 NXB XIC N40:0/2 XIC N11:9/0 SCP N40:5 0 15 120 90 N7:90 BND NXB XIO B3:9/8 MOV 105 N7:90 NXB BST XIC B3:14/4 NXB XIC B3:14/5 BND SCP N40:7 0 15 120 90 N7:90 NXB BST MOV 200 T4:92.PRE NXB XIC B3:9/8 BST XIC B3:12/12 XIO B3:14/9 BST OTE B3:14/8 NXB TON T4:92 0.01 200 0 BND NXB BST XIC T4:92/DN NXB XIC B3:14/9 BND OTE B3:14/9 BND BND BND EOR
%   B3:9/8  WRAPMEMORY  "Wrap Load Memory" %
%   B3:14/4  "Metered Pre-Stretch Payout For Film Cut" %
%   N40:0/1  "Current Profile Force Bottom Enable" %
%   N11:13/1  CARRIAGEDOWN  "- Input - Film Carriage Down" %
%   N40:6  "Current Profile Force At Bottom" %
%   N7:90  "Metered Pre-Stretch Current Payout (100 = 100%)" %
%   N40:0/2  "Current Profile Force Top Enable" %
%   N11:9/0  HEIGHTSENSING  "- Input - Load Height Sensing Clear" %
%   N40:8  "Current Profile Force At Load" %
%   N40:5  "Current Profile Force At Top" %
%   B3:14/5  "Metered Pre-Stretch Payout For Film Clamp" %
%   N40:7  "Current Profile Force During Cut" %
%   T4:92  "Metered Pre-Stretch Starting Payout Complete Delay" %
%   B3:12/12  ROTATIONRUNNING  "Rotation Running" %
%   B3:14/9  "Metered Pre-Stretch Starting Payout Complete" %
%   B3:14/8  "Metered Pre-Stretch Starting Payout" %

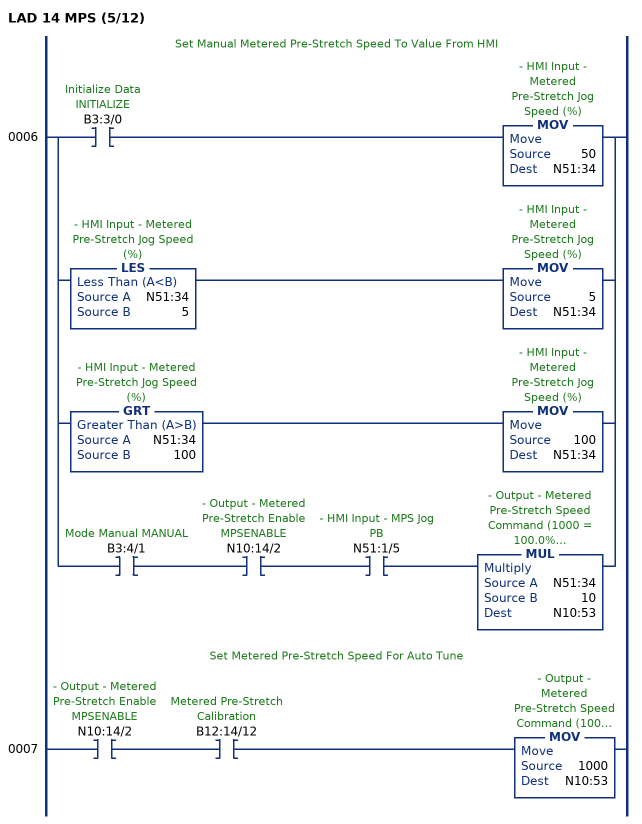
% Rung: 6 %
% Set Manual Metered Pre-Stretch Speed To Value From HMI %
SOR BST BST XIC B3:3/0 MOV 50 N51:34 NXB LES N51:34 5 MOV 5 N51:34 NXB GRT N51:34 100 MOV 100 N51:34 BND NXB XIC B3:4/1 XIC N10:14/2 XIC N51:1/5 MUL N51:34 10 N10:53 BND EOR
%   B3:3/0  INITIALIZE  "Initialize Data" %
%   N51:34  "- HMI Input - Metered Pre-Stretch Jog Speed (%)" %
%   B3:4/1  MANUAL  "Mode Manual" %
%   N10:14/2  MPSENABLE  "- Output - Metered Pre-Stretch Enable" %
%   N51:1/5  "- HMI Input - MPS Jog PB" %
%   N10:53  MPSCOMMAND  "- Output - Metered Pre-Stretch Speed Command (1000 = 100.0%)" %
% Rung: 7 %
% Set Metered Pre-Stretch Speed For Auto Tune %
SOR XIC N10:14/2 XIC B12:14/12 MOV 1000 N10:53 EOR
%   N10:14/2  MPSENABLE  "- Output - Metered Pre-Stretch Enable" %
%   B12:14/12  "Metered Pre-Stretch Calibration" %
%   N10:53  MPSCOMMAND  "- Output - Metered Pre-Stretch Speed Command (1000 = 100.0%)" %

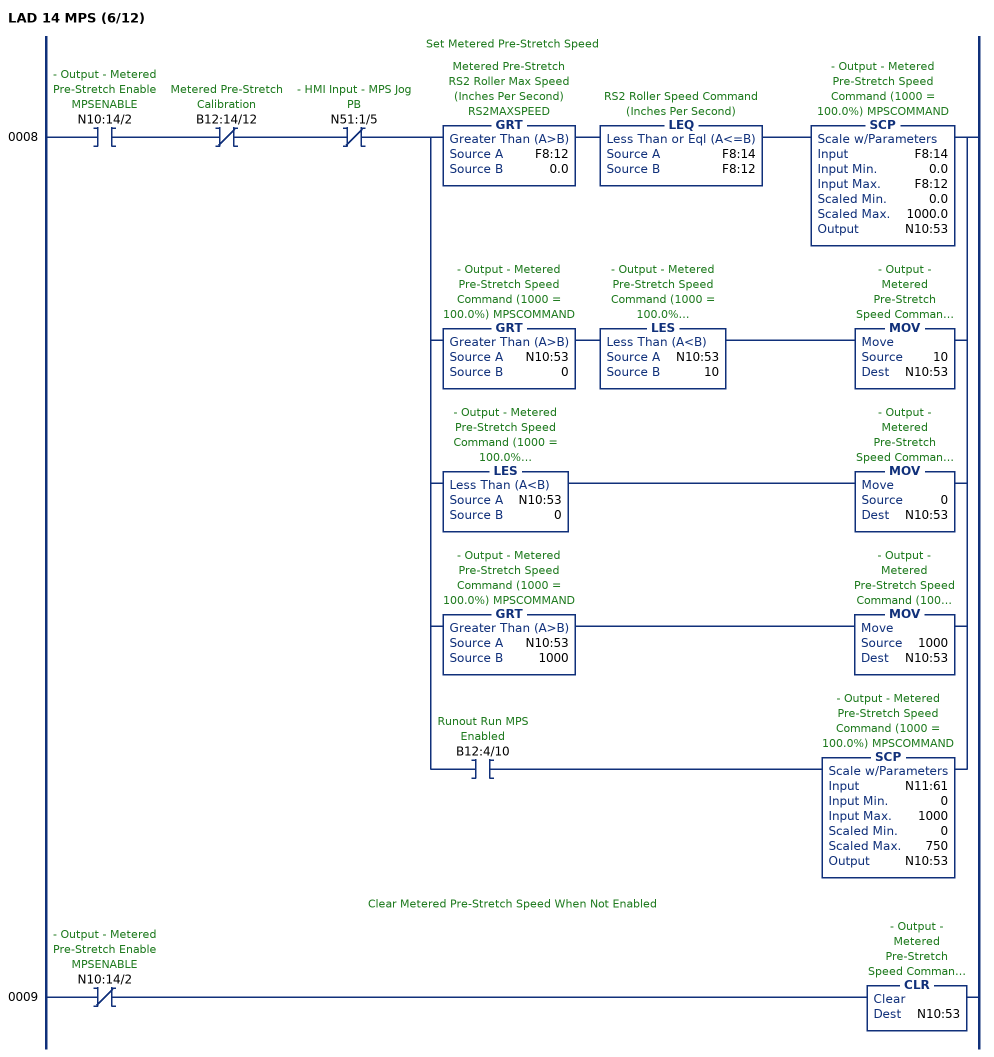
% Rung: 8 %
% Set Metered Pre-Stretch Speed %
SOR XIC N10:14/2 XIO B12:14/12 XIO N51:1/5 BST GRT F8:12 0.0 LEQ F8:14 F8:12 SCP F8:14 0.0 F8:12 0.0 1000.0 N10:53 NXB GRT N10:53 0 LES N10:53 10 MOV 10 N10:53 NXB LES N10:53 0 MOV 0 N10:53 NXB GRT N10:53 1000 MOV 1000 N10:53 NXB XIC B12:4/10 SCP N11:61 0 1000 0 750 N10:53 BND EOR
%   N10:14/2  MPSENABLE  "- Output - Metered Pre-Stretch Enable" %
%   B12:14/12  "Metered Pre-Stretch Calibration" %
%   N51:1/5  "- HMI Input - MPS Jog PB" %
%   F8:12  RS2MAXSPEED  "Metered Pre-Stretch RS2 Roller Max Speed (Inches Per Second)" %
%   F8:14  "RS2 Roller Speed Command (Inches Per Second)" %
%   N10:53  MPSCOMMAND  "- Output - Metered Pre-Stretch Speed Command (1000 = 100.0%)" %
%   B12:4/10  "Runout Run MPS Enabled" %
%   N11:61  "- Input - Rotation VFD Speed Feedback" %
% Rung: 9 %
% Clear Metered Pre-Stretch Speed When Not Enabled %
SOR XIO N10:14/2 CLR N10:53 EOR
%   N10:14/2  MPSENABLE  "- Output - Metered Pre-Stretch Enable" %
%   N10:53  MPSCOMMAND  "- Output - Metered Pre-Stretch Speed Command (1000 = 100.0%)" %

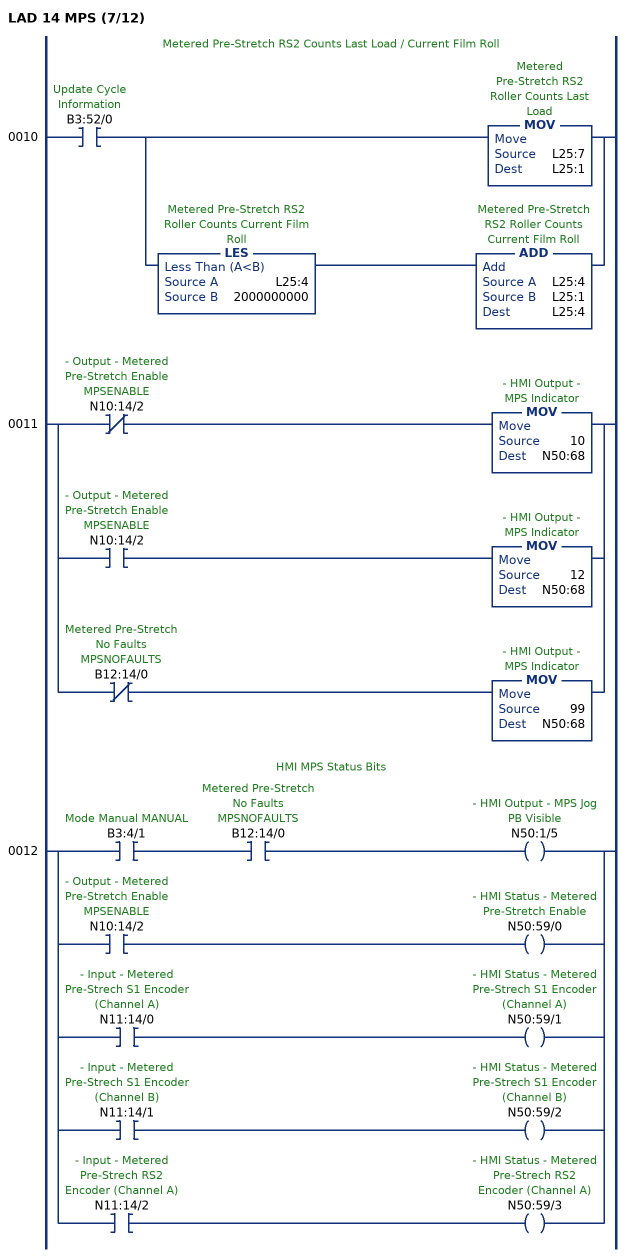
% Rung: 10 %
% Metered Pre-Stretch RS2 Counts Last Load / Current Film Roll %
SOR XIC B3:52/0 BST MOV L25:7 L25:1 NXB LES L25:4 2000000000 ADD L25:4 L25:1 L25:4 BND EOR
%   B3:52/0  "Update Cycle Information" %
%   L25:7  "Metered Pre-Stretch RS2 Roller Current Count" %
%   L25:1  "Metered Pre-Stretch RS2 Roller Counts Last Load" %
%   L25:4  "Metered Pre-Stretch RS2 Roller Counts Current Film Roll" %
% Rung: 11 %
SOR BST XIO N10:14/2 MOV 10 N50:68 NXB XIC N10:14/2 MOV 12 N50:68 NXB XIO B12:14/0 MOV 99 N50:68 BND EOR
%   N10:14/2  MPSENABLE  "- Output - Metered Pre-Stretch Enable" %
%   N50:68  "- HMI Output - MPS Indicator" %
%   B12:14/0  MPSNOFAULTS  "Metered Pre-Stretch No Faults" %
% Rung: 12 %
% HMI MPS Status Bits %
SOR BST XIC B3:4/1 XIC B12:14/0 OTE N50:1/5 NXB XIC N10:14/2 OTE N50:59/0 NXB XIC N11:14/0 OTE N50:59/1 NXB XIC N11:14/1 OTE N50:59/2 NXB XIC N11:14/2 OTE N50:59/3 BND EOR
%   B3:4/1  MANUAL  "Mode Manual" %
%   B12:14/0  MPSNOFAULTS  "Metered Pre-Stretch No Faults" %
%   N50:1/5  "- HMI Output - MPS Jog PB Visible" %
%   N10:14/2  MPSENABLE  "- Output - Metered Pre-Stretch Enable" %
%   N50:59/0  "- HMI Status - Metered Pre-Stretch Enable" %
%   N11:14/0  "- Input - Metered Pre-Strech S1 Encoder (Channel A)" %
%   N50:59/1  "- HMI Status - Metered Pre-Strech S1 Encoder (Channel A)" %
%   N11:14/1  "- Input - Metered Pre-Strech S1 Encoder (Channel B)" %
%   N50:59/2  "- HMI Status - Metered Pre-Strech S1 Encoder (Channel B)" %
%   N11:14/2  "- Input - Metered Pre-Strech RS2 Encoder (Channel A)" %
%   N50:59/3  "- HMI Status - Metered Pre-Strech RS2 Encoder (Channel A)" %

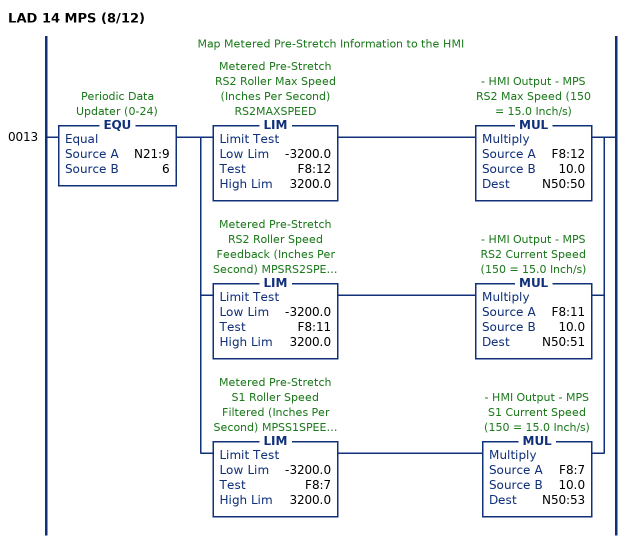
% Rung: 13 %
% Map Metered Pre-Stretch Information to the HMI %
SOR EQU N21:9 6 BST LIM -3200.0 F8:12 3200.0 MUL F8:12 10.0 N50:50 NXB LIM -3200.0 F8:11 3200.0 MUL F8:11 10.0 N50:51 NXB LIM -3200.0 F8:7 3200.0 MUL F8:7 10.0 N50:53 BND EOR
%   N21:9  "Periodic Data Updater (0-24)" %
%   F8:12  RS2MAXSPEED  "Metered Pre-Stretch RS2 Roller Max Speed (Inches Per Second)" %
%   N50:50  "- HMI Output - MPS RS2 Max Speed (150 = 15.0 Inch/s)" %
%   F8:11  MPSRS2SPEED  "Metered Pre-Stretch RS2 Roller Speed Feedback (Inches Per Second)" %
%   N50:51  "- HMI Output - MPS RS2 Current Speed (150 = 15.0 Inch/s)" %
%   F8:7  MPSS1SPEEDFILTERED  "Metered Pre-Stretch S1 Roller Speed Filtered (Inches Per Second)" %
%   N50:53  "- HMI Output - MPS S1 Current Speed (150 = 15.0 Inch/s)" %

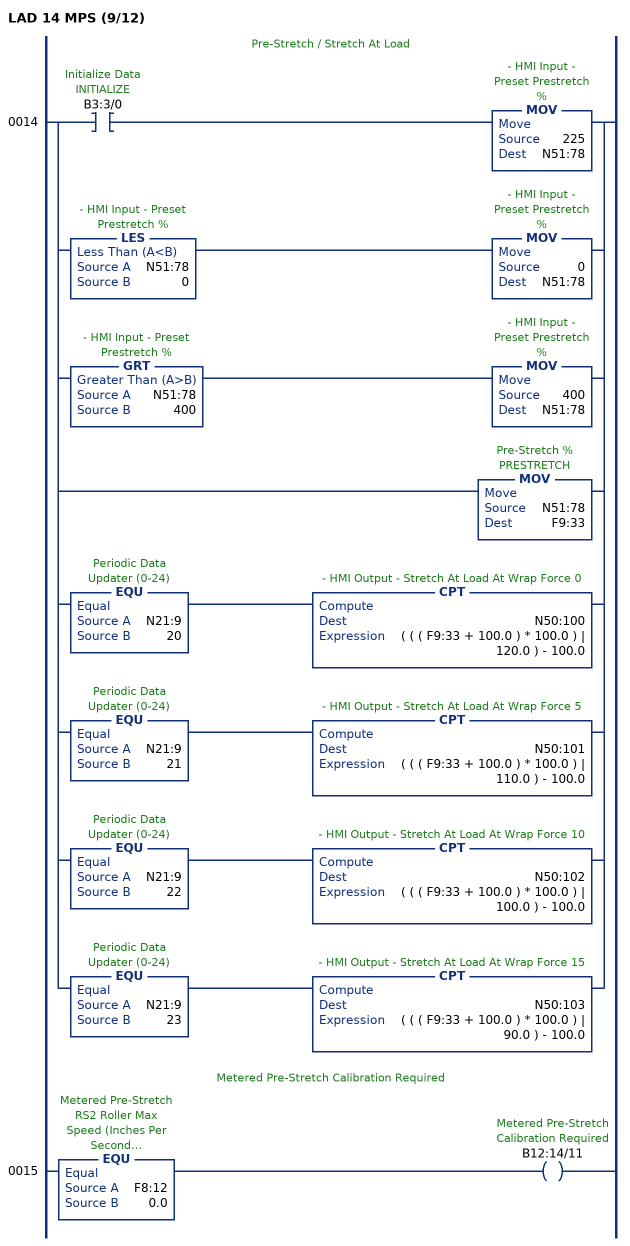
% Rung: 14 %
% Pre-Stretch / Stretch At Load %
SOR BST BST XIC B3:3/0 MOV 225 N51:78 NXB LES N51:78 0 MOV 0 N51:78 NXB GRT N51:78 400 MOV 400 N51:78 NXB MOV N51:78 F9:33 BND NXB EQU N21:9 20 CPT N50:100 " ( ( ( F9:33 + 100.0 ) * 100.0 ) | 120.0 ) - 100.0 " NXB EQU N21:9 21 CPT N50:101 " ( ( ( F9:33 + 100.0 ) * 100.0 ) | 110.0 ) - 100.0 " NXB EQU N21:9 22 CPT N50:102 " ( ( ( F9:33 + 100.0 ) * 100.0 ) | 100.0 ) - 100.0 " NXB EQU N21:9 23 CPT N50:103 " ( ( ( F9:33 + 100.0 ) * 100.0 ) | 90.0 ) - 100.0 " BND EOR
%   B3:3/0  INITIALIZE  "Initialize Data" %
%   N51:78  "- HMI Input - Preset Prestretch %" %
%   F9:33  PRESTRETCH  "Pre-Stretch %" %
%   N21:9  "Periodic Data Updater (0-24)" %
%   N50:100  "- HMI Output - Stretch At Load At Wrap Force 0" %
%   N50:101  "- HMI Output - Stretch At Load At Wrap Force 5" %
%   N50:102  "- HMI Output - Stretch At Load At Wrap Force 10" %
%   N50:103  "- HMI Output - Stretch At Load At Wrap Force 15" %
% Rung: 15 %
% Metered Pre-Stretch Calibration Required %
SOR EQU F8:12 0.0 OTE B12:14/11 EOR
%   F8:12  RS2MAXSPEED  "Metered Pre-Stretch RS2 Roller Max Speed (Inches Per Second)" %
%   B12:14/11  "Metered Pre-Stretch Calibration Required" %

